(* IEC 61131-3 sources: Elmo_Master/Lasal_PRG/MotionTCPDemo/Class/_LMCModuleBase, 1 file *)

(* ---- _LMCModuleBase.st ---- *)
(*!
<Class
	Name               = "_LMCModuleBase"
	Revision           = "1.1"
	RealtimeTask       = "false"
	CyclicTask         = "false"
	BackgroundTask     = "false"
	Sigmatek           = "true"
	OSInterface        = "false"
	HighPriority       = "false"
	Automatic          = "false"
	UpdateMode         = "Prescan"
	IconPath           = ".\Class\_AxisBase\LMCAxis.ico"
	SharedCommandTable = "true"
	Objectsize         = "(480,120)"
	Comment            = "derive this class to implement user defined calculations">
	<Channels>
		<Server Name="ClassSvr" Visualized="false" Initialize="false" WriteProtected="false" Retentive="false" Comment=" 0 ... login was successful&#13;&#10;-1 ... index out of range"/>
		<Client Name="_LMCAxis" Required="true" Internal="false" Comment="objectchannel "/>
		<Client Name="Config" Required="false" Internal="false" Comment="0 ... position-offset&#13;&#10;10 ... PreRtWork&#13;&#10;11 ... PostRtWork"/>
		<Client Name="Index" Required="false" Internal="false" Comment="calling order"/>
	</Channels>
	<RevDoku>
		<Owner Company="Sigmatek" Author="HasHan"/>
		<Dokumentation Revision="1.1" Date="2024-06-17" Author="StePhi" Company="Sigmatek" Description="Bugfix: Return values of NewInst with uiCmd-Index 0 and 1 to manipulate ActPos and SetPos fixed."/>
		<Dokumentation Revision="1.0" Date="2019-03-04" Author="HasHan" Company="Sigmatek" Description="creation"/>
	</RevDoku>
</Class>
*)
_LMCModuleBase : CLASS
  //Servers:
	ClassSvr 	: SvrChCmd_DINT;
  //Clients:
	_LMCAxis 	: CltChCmd__LMCAxisBase;
	Index 	: CltCh_DINT;
	Config 	: CltCh_DINT;
  //Variables:
		pCNCVars 	: ^CNCInternalStruct;
  //Functions:

	FUNCTION VIRTUAL GLOBAL Init;

	FUNCTION VIRTUAL GLOBAL ClassSvr::NewInst
		VAR_INPUT
			pPara 	: ^CmdStruct;
			pResult 	: ^results;
		END_VAR
		VAR_OUTPUT
			ret_code 	: iprStates;
		END_VAR;
  //Tables:
	FUNCTION @STD
		VAR_OUTPUT
			ret_code	: CONFSTATES;
		END_VAR;
	FUNCTION GLOBAL TAB @CT_;
END_CLASS;

#pragma usingLtd _LMCAxisBase

FUNCTION VIRTUAL GLOBAL _LMCModuleBase::Init

  if _FirstScan then
    if IsClientConnected(#_LMCAxis) = 1 then
      ClassSvr := _LMCAxis.Login(this, Index, Config);
    end_if;
  end_if;

END_FUNCTION

FUNCTION VIRTUAL GLOBAL _LMCModuleBase::ClassSvr::NewInst
	VAR_INPUT
		pPara 	: ^CmdStruct;
		pResult 	: ^results;
	END_VAR
	VAR_OUTPUT
		ret_code 	: iprStates;
	END_VAR

  ret_code := BUSY;

  case pPara^.uiCmd of
    //******************************************************************************************************
    0: //BinAct manipulation
    //******************************************************************************************************
      pResult^.aData$DINT := 0;
      ret_code := READY;

    //******************************************************************************************************
    1: //TrapPosAct/RoundPosAct manipulation
    //******************************************************************************************************
      pResult^.aData$DINT := 0;
      ret_code := READY;

    //******************************************************************************************************
    10: //PreRtWork
    //******************************************************************************************************
      pResult^.aData$DINT := pPara^.aPara[0];
      ret_code := READY;

    //******************************************************************************************************
    11: //PostRtWork
    //******************************************************************************************************
      pResult^.aData$DINT := pPara^.aPara[0];
      ret_code := READY;

  end_case;

END_FUNCTION
